DATA_BLOCK "DI_Host_Recv_Ext_T"
TITLE =%version: 0.02 % CN: 49
//History:
//This version  %created_by: nlhdl %
//              %date_created: maandag 6 juli 2015 10:44:01 %
//
//Modification History:                                   By:    Date:     Rev:
//----------------------------------------------------  -------  --------  -----
//7324: ECS-P General from the RD to RA for platform    nlHdL    06-07-15   0.02
FAMILY : VIBES
VERSION : 0.0

"FB_Host_Recv_Ext_T"
BEGIN
END_DATA_BLOCK
